(* LS Electric XG5000 project: 23_10_31 *)
(* PLC LSPLC *)

PROGRAM NewProgram (* task: 스캔 프로그램 *)
VAR
    in1 : BOOL;
    INST1 : TON;
    INST2 : TON;
    Q10_P1 : BOOL;
    Q10_P10 : BOOL;
    Q10_t1 : TON;
    Q10_t2 : TON;
    Q10_t3 : TOF;
    Q10_t4 : TON;
    Q11_P1 : BOOL;
    Q11_P10 : BOOL;
    Q11_P11 : BOOL;
    Q11_P12 : BOOL;
    Q11_tp1 : TP;
    Q11_tp2 : TP;
    Q11_tp3 : TP;
    Q12_ctu : CTU_INT;
    Q12_P1 : BOOL;
    Q12_P10 : BOOL;
    Q12_P2 : BOOL;
    Q13_ctu1 : CTU_INT;
    Q13_ctu2 : CTU_INT;
    Q13_ctu3 : CTU_INT;
    Q13_P1 : BOOL;
    Q13_P10 : BOOL;
    Q13_P11 : BOOL;
    r : BOOL;
END_VAR

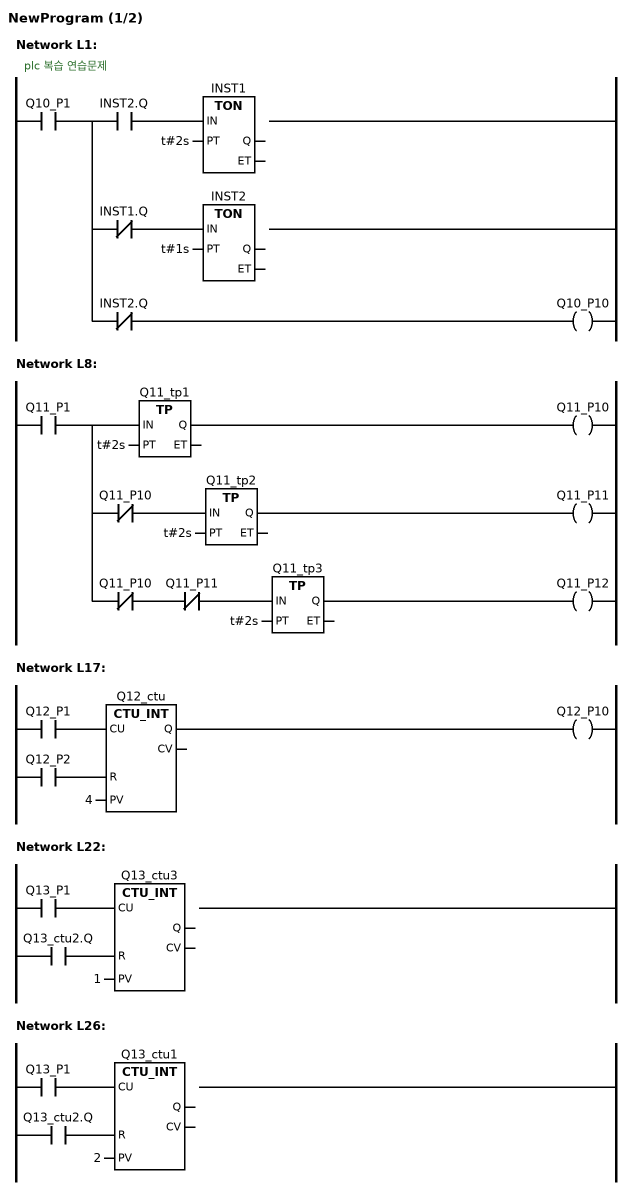
(* plc 복습 연습문제 *)
(* Rung L1 *)
INST1(IN := Q10_P1 AND INST2.Q, PT := t#2s);
INST2(IN := Q10_P1 AND NOT INST1.Q, PT := t#1s);
Q10_P10 := Q10_P1 AND NOT INST2.Q;
(* Rung L8 *)
Q11_tp1(IN := Q11_P1, PT := t#2s);
Q11_P10 := Q11_tp1.Q;
Q11_tp2(IN := Q11_P1 AND NOT Q11_P10, PT := t#2s);
Q11_P11 := Q11_tp2.Q;
Q11_tp3(IN := Q11_P1 AND NOT Q11_P10 AND NOT Q11_P11, PT := t#2s);
Q11_P12 := Q11_tp3.Q;
(* Rung L17 *)
Q12_ctu(CU := Q12_P1, R := Q12_P2, PV := 4);
Q12_P10 := Q12_ctu.Q;
(* Rung L22 *)
Q13_ctu3(CU := Q13_P1, R := Q13_ctu2.Q, PV := 1);
(* Rung L26 *)
Q13_ctu1(CU := Q13_P1, R := Q13_ctu2.Q, PV := 2);

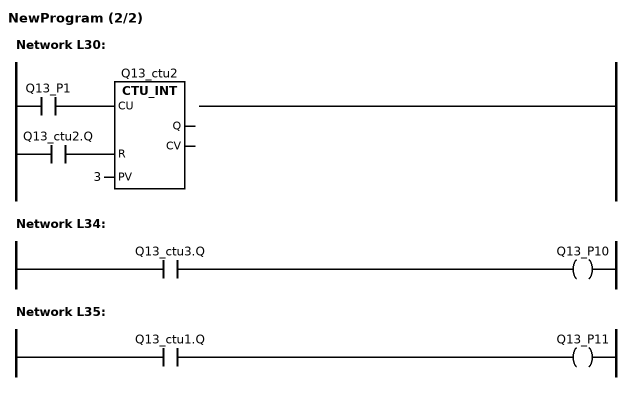
(* Rung L30 *)
Q13_ctu2(CU := Q13_P1, R := Q13_ctu2.Q, PV := 3);
(* Rung L34 *)
Q13_P10 := Q13_ctu3.Q;
(* Rung L35 *)
Q13_P11 := Q13_ctu1.Q;
END_PROGRAM